(* CoDeSys 2.3.9.418 project: testApp.pro *)
(* Libraries: Util.lib 18.5.10 15:14:28, STANDARD.LIB 4.10.05 11:14:46, IECSFC.LIB 13.4.06 15:51:28, SYSLIBTIME.LIB 6.11.19 15:29:28, ANALYZATION.LIB 5.10.99 09:05:06 *)

(* PLC configuration (modules and I/O channels)
Fast discrete inputs [I_SIMPLE_INPUT] node 0, in %IB0 out %QB0 {Filtrationtime = 10}
  AT %IX0.0 [BitInput] Discrete input 1
  AT %IX0.1 [BitInput] Discrete input 2
  AT %IX0.2 [BitInput] Discrete input 3
  AT %IX0.3 [BitInput] Discrete input 4
Discrete inputs [ID130] node 1, in %IB1 out %QB1 {Filtrationtime_GeneralINP = 10; Visibility = No; PinCount = 12}
  AT %IB1.0 [ByteInput] 8 discrete inputs
  AT %IB1.1 [ByteInput] 4 discrete inputs
Discrete outputs [ID131] node 2, in %IB2 out %QB2 {SafeValueByte = 0; SafeValueByteM = 0; Visibility = No; PinCount = 12}
  AT %QB2.0 [ByteOutput] 8 discrete outputs
  AT %QB2.1 [ByteOutput] 4 discrete outputs
Fast analog inputs [ID125] node 3, in %IB3 out %QB3 {Flt_Comm = 50Hz 2Por}
  AT %IR3.0 [FloatInputP] AI #1 {AIN_TYPE = 4-20 mA; Peak_Filtr = 200; Flt_Ch = Off; TauRC = 10; MinFV = 0; MaxFV = 20000.0}
  AT %IR3.1 [FloatInputP] AI #2 {AIN_TYPE = 4-20 mA; Peak_Filtr = 200; Flt_Ch = Off; TauRC = 10; MinFV = 0; MaxFV = 20000.0}
  AT %IR3.2 [FloatInputP] AI #3 {AIN_TYPE = 4-20 mA; Peak_Filtr = 200; Flt_Ch = Off; TauRC = 10; MinFV = 0; MaxFV = 20000.0}
  AT %IR3.3 [FloatInputP] AI #4 {AIN_TYPE = 4-20 mA; Peak_Filtr = 200; Flt_Ch = Off; TauRC = 10; MinFV = 0; MaxFV = 20000.0}
  AT %IR3.4 [FloatInputP] AI #5 {AIN_TYPE = 4-20 mA; Peak_Filtr = 200; Flt_Ch = Off; TauRC = 10; MinFV = 0; MaxFV = 20000.0}
  AT %IR3.5 [FloatInputP] AI #6 {AIN_TYPE = 4-20 mA; Peak_Filtr = 200; Flt_Ch = Off; TauRC = 10; MinFV = 0; MaxFV = 20000.0}
  AT %IR3.6 [FloatInputP] AI #7 {AIN_TYPE = 4-20 mA; Peak_Filtr = 200; Flt_Ch = Off; TauRC = 10; MinFV = 0; MaxFV = 20000.0}
  AT %IR3.7 [FloatInputP] AI #8 {AIN_TYPE = 4-20 mA; Peak_Filtr = 200; Flt_Ch = Off; TauRC = 10; MinFV = 0; MaxFV = 20000.0}
  AT %IW3.8 [WordInput] AI read time (10ms)
Analog outputs [ID126] node 4, in %IB4 out %QB4
  AT %QR4.0 [FloatOutputP] AO #1 {AOUT_TYPE = 4-20 mA; SafeValueREAL = 0.0}
  AT %QR4.1 [FloatOutputP] AO #2 {AOUT_TYPE = 4-20 mA; SafeValueREAL = 0.0}
  AT %QR4.2 [FloatOutputP] AO #3 {AOUT_TYPE = 4-20 mA; SafeValueREAL = 0.0}
  AT %QR4.3 [FloatOutputP] AO #4 {AOUT_TYPE = 4-20 mA; SafeValueREAL = 0.0}
Special input [ID103] node 5, in %IB5 out %QB5 {Filtrationtime = 1000; PinCount = 1; WatchDogPeriod = 400; PollPeriod = 3000; Visibility = No}
  AT %IX5.0 [BitInput] Special input
Special output [ID104] node 6, in %IB6 out %QB6 {Visibility = No; PinCount = 1}
  AT %QX6.0 [BitOutput] Special output
ModBus (Master) [MODBUS_MASTER_ID450] node 7, in %IB7 out %QB7 {Visibility = No}
  AT %QD7.0 [DWordOutput] Last address
  AT %QW7.1 [WordOutput] Last error
  RS-485-1 [COM1_USART] node 0, in %IB7.0 out %QB7.0 {CommunicationSpeed = 57600; Parity = NO PARITY CHECK; BitLength = 8 bits; StopLength = One stop bit; InterfaceType = RS485; FrameOriented = RTU; Timeout = 0; Visibility = No}
AT %QB7.1.0 [ComChannel] Command (0xff - Start)
addAO0 AT %QW7.1.0.0 [WordOutput]
addAO1 AT %QW7.1.1.0 [WordOutput]
AT %QB7.2.0 [ComChannel] Command (0xff - Start)
addDI AT %ID7.2.0.0 [DWordInput]
AT %QB7.3.0 [ComChannel] Command (0xff - Start)
addDO AT %QD7.3.0.0 [DWordOutput]
AT %QD8.0 [DWordOutput] Last address
AT %QW8.1 [WordOutput] Last error
RS-232 [COM2_USART] node 0, in %IB8.0 out %QB8.0 {CommunicationSpeed = 57600; Parity = NO PARITY CHECK; BitLength = 8 bits; StopLength = One stop bit; InterfaceType = RS232; FrameOriented = RTU; Timeout = 0; Visibility = No}
AT %QB8.1.0 [ComChannel] Command (0xff - Start)
8 bit input module [ID2001] node 0, in %IB8.1.0 out %QB8.1.0 {ModbusAddress = 256; Command_read_byte = Read coils status (0x01); Visibility = No}
  AT %IB8.1.0.0 [ByteInput]
8 bit input module [ID2001] node 1, in %IB8.1.1 out %QB8.1.1 {ModbusAddress = 264; Command_read_byte = Read coils status (0x01); Visibility = No}
  AT %IB8.1.1.0 [ByteInput]
panInTestWord0 AT %IW8.1.2.0 [WordInput]
panSetAO0 AT %ID8.1.3.0 [FloatInput]
panSetAO1 AT %ID8.1.4.0 [FloatInput]
AT %QB8.2.0 [ComChannel] Command (0xff - Start)
8 bit output module [ID2002] node 0, in %IB8.2.0 out %QB8.2.0 {ModbusAddress = 272; Command_write_byte = Force multiply coils (0x0f); Visibility = No}
  AT %QB8.2.0.0 [ByteOutput]
8 bit output module [ID2002] node 1, in %IB8.2.1 out %QB8.2.1 {ModbusAddress = 280; Command_write_byte = Force multiply coils (0x0f); Visibility = No}
  AT %QB8.2.1.0 [ByteOutput]
panOutTestWord0 AT %QW8.2.2.0 [WordOutput]
AT %QD8.2.3.0 [FloatOutput]
*)

(* POU PLC_PRG, CFC *)
PROGRAM PLC_PRG
VAR
	blink_0: BLINK;
	blink_1: BLINK;
	blink_2: BLINK;
	blink_3: BLINK;
	blink_4: BLINK;
	blink_5: BLINK;
	blink_6: BLINK;
	blink_7: BLINK;
	blink_8: BLINK;
	blink_9: BLINK;
	blink_10: BLINK;
	blink_11: BLINK;
	startBlink0: BOOL;
	startBlink1: BOOL;
	startBlink2: BOOL;
	startBlink3: BOOL;
	startBlink4: BOOL;
	startBlink5: BOOL;
	startBlink6: BOOL;
	startBlink7: BOOL;
	startBlink8: BOOL;
	startBlink9: BOOL;
	startBlink10: BOOL;
	startBlink11: BOOL;
	gen_0: GEN;
	genOut: INT;
	setAmpl: INT;

	addDIblink: BLINK;
END_VAR
VAR (* helpers for the ST form of the networks *)
	_t183 : WORD;
	_t189 : WORD;
END_VAR
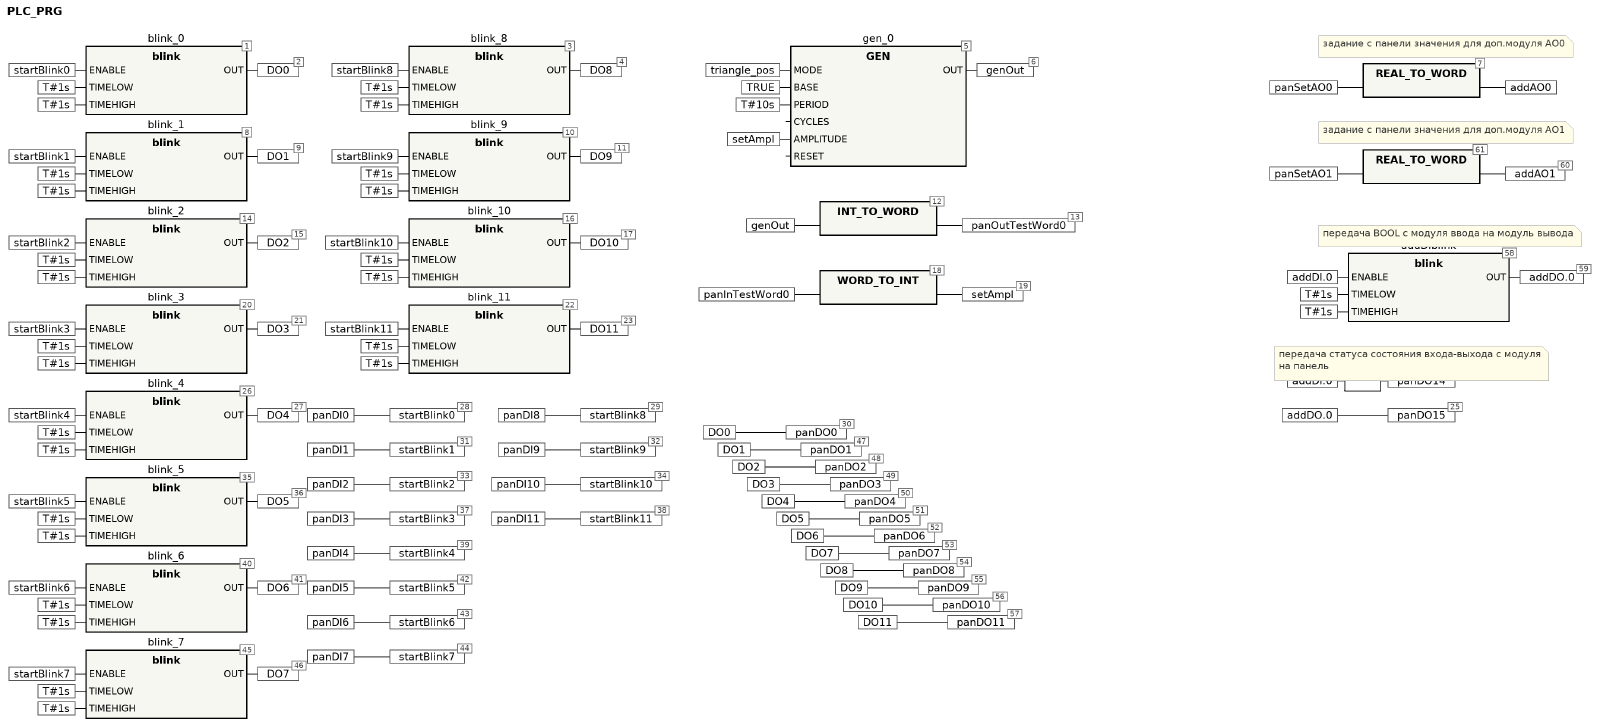
_CFC_ (* Continuous Function Chart, elements in execution order *)
(* задание с панели значения для доп.модуля AO0 *)
#0 addAO0 <= #7
#1 blink_0:blink(ENABLE: startBlink0, TIMELOW: T#1s, TIMEHIGH: T#1s)
#2 DO0 <= #1.OUT
#3 blink_8:blink(ENABLE: startBlink8, TIMELOW: T#1s, TIMEHIGH: T#1s)
#4 DO8 <= #3.OUT
#5 gen_0:GEN(MODE: triangle_pos, BASE: TRUE, PERIOD: T#10s, CYCLES: -, AMPLITUDE: setAmpl, RESET: -)
#6 genOut <= #5.OUT
#7 REAL_TO_WORD(panSetAO0)
#8 blink_1:blink(ENABLE: startBlink1, TIMELOW: T#1s, TIMEHIGH: T#1s)
#9 DO1 <= #8.OUT
#10 blink_9:blink(ENABLE: startBlink9, TIMELOW: T#1s, TIMEHIGH: T#1s)
#11 DO9 <= #10.OUT
#12 INT_TO_WORD(genOut)
#13 panOutTestWord0 <= #12
#14 blink_2:blink(ENABLE: startBlink2, TIMELOW: T#1s, TIMEHIGH: T#1s)
#15 DO2 <= #14.OUT
#16 blink_10:blink(ENABLE: startBlink10, TIMELOW: T#1s, TIMEHIGH: T#1s)
#17 DO10 <= #16.OUT
#18 WORD_TO_INT(panInTestWord0)
#19 setAmpl <= #18
#20 blink_3:blink(ENABLE: startBlink3, TIMELOW: T#1s, TIMEHIGH: T#1s)
#21 DO3 <= #20.OUT
#22 blink_11:blink(ENABLE: startBlink11, TIMELOW: T#1s, TIMEHIGH: T#1s)
#23 DO11 <= #22.OUT
#24 panDO14 <= addDI.0
#25 panDO15 <= addDO.0
#26 blink_4:blink(ENABLE: startBlink4, TIMELOW: T#1s, TIMEHIGH: T#1s)
#27 DO4 <= #26.OUT
#28 startBlink0 <= panDI0
#29 startBlink8 <= panDI8
#30 panDO0 <= DO0
#31 startBlink1 <= panDI1
#32 startBlink9 <= panDI9
#33 startBlink2 <= panDI2
#34 startBlink10 <= panDI10
#35 blink_5:blink(ENABLE: startBlink5, TIMELOW: T#1s, TIMEHIGH: T#1s)
#36 DO5 <= #35.OUT
#37 startBlink3 <= panDI3
#38 startBlink11 <= panDI11
#39 startBlink4 <= panDI4
#40 blink_6:blink(ENABLE: startBlink6, TIMELOW: T#1s, TIMEHIGH: T#1s)
#41 DO6 <= #40.OUT
#42 startBlink5 <= panDI5
#43 startBlink6 <= panDI6
#44 startBlink7 <= panDI7
#45 blink_7:blink(ENABLE: startBlink7, TIMELOW: T#1s, TIMEHIGH: T#1s)
#46 DO7 <= #45.OUT
#47 panDO1 <= DO1
#48 panDO2 <= DO2
#49 panDO3 <= DO3
#50 panDO4 <= DO4
#51 panDO5 <= DO5
#52 panDO6 <= DO6
#53 panDO7 <= DO7
#54 panDO8 <= DO8
#55 panDO9 <= DO9
#56 panDO10 <= DO10
#57 panDO11 <= DO11
#58 addDIblink:blink(ENABLE: addDI.0, TIMELOW: T#1s, TIMEHIGH: T#1s)
#59 addDO.0 <= #58.OUT
(* передача BOOL с модуля ввода на модуль вывода *)
(* передача статуса состояния входа-выхода с модуля на панель *)
(* задание с панели значения для доп.модуля AO1 *)
#60 addAO1 <= #61
#61 REAL_TO_WORD(panSetAO1)
_END_CFC_
(* the same logic as Structured Text *)
(* задание с панели значения для доп.модуля AO0 *)
addAO0 := _t183;
blink_0(ENABLE := startBlink0, TIMELOW := T#1s, TIMEHIGH := T#1s);
DO0 := blink_0.OUT;
blink_8(ENABLE := startBlink8, TIMELOW := T#1s, TIMEHIGH := T#1s);
DO8 := blink_8.OUT;
gen_0(MODE := triangle_pos, BASE := TRUE, PERIOD := T#10s, AMPLITUDE := setAmpl);
genOut := gen_0.OUT;
_t183 := REAL_TO_WORD(panSetAO0);
blink_1(ENABLE := startBlink1, TIMELOW := T#1s, TIMEHIGH := T#1s);
DO1 := blink_1.OUT;
blink_9(ENABLE := startBlink9, TIMELOW := T#1s, TIMEHIGH := T#1s);
DO9 := blink_9.OUT;
panOutTestWord0 := INT_TO_WORD(genOut);
blink_2(ENABLE := startBlink2, TIMELOW := T#1s, TIMEHIGH := T#1s);
DO2 := blink_2.OUT;
blink_10(ENABLE := startBlink10, TIMELOW := T#1s, TIMEHIGH := T#1s);
DO10 := blink_10.OUT;
setAmpl := WORD_TO_INT(panInTestWord0);
blink_3(ENABLE := startBlink3, TIMELOW := T#1s, TIMEHIGH := T#1s);
DO3 := blink_3.OUT;
blink_11(ENABLE := startBlink11, TIMELOW := T#1s, TIMEHIGH := T#1s);
DO11 := blink_11.OUT;
panDO14 := addDI.0;
panDO15 := addDO.0;
blink_4(ENABLE := startBlink4, TIMELOW := T#1s, TIMEHIGH := T#1s);
DO4 := blink_4.OUT;
startBlink0 := panDI0;
startBlink8 := panDI8;
panDO0 := DO0;
startBlink1 := panDI1;
startBlink9 := panDI9;
startBlink2 := panDI2;
startBlink10 := panDI10;
blink_5(ENABLE := startBlink5, TIMELOW := T#1s, TIMEHIGH := T#1s);
DO5 := blink_5.OUT;
startBlink3 := panDI3;
startBlink11 := panDI11;
startBlink4 := panDI4;
blink_6(ENABLE := startBlink6, TIMELOW := T#1s, TIMEHIGH := T#1s);
DO6 := blink_6.OUT;
startBlink5 := panDI5;
startBlink6 := panDI6;
startBlink7 := panDI7;
blink_7(ENABLE := startBlink7, TIMELOW := T#1s, TIMEHIGH := T#1s);
DO7 := blink_7.OUT;
panDO1 := DO1;
panDO2 := DO2;
panDO3 := DO3;
panDO4 := DO4;
panDO5 := DO5;
panDO6 := DO6;
panDO7 := DO7;
panDO8 := DO8;
panDO9 := DO9;
panDO10 := DO10;
panDO11 := DO11;
addDIblink(ENABLE := addDI.0, TIMELOW := T#1s, TIMEHIGH := T#1s);
addDO.0 := addDIblink.OUT;
(* передача BOOL с модуля ввода на модуль вывода *)
(* передача статуса состояния входа-выхода с модуля на панель *)
(* задание с панели значения для доп.модуля AO1 *)
addAO1 := _t189;
_t189 := REAL_TO_WORD(panSetAO1);
END_PROGRAM
